// TIA Portal V16 export
// export: Created 2022-08-05T16:49:58.9120399Z, ExportSetting WithDefaults, DisplayName Totally Integrated Automation Portal, DisplayVersion V16, DisplayName TIA Portal Version Control Interface, DisplayVersion V16, DisplayName TIA Portal Openness, DisplayVersion V16, DisplayName SINAMICS Startdrive Advanced, DisplayVersion V16, DisplayName SINAMICS Startdrive G130, G150, S120, S150, SINAMICS MV, S210, DisplayVersion V16, DisplayName SINAMICS Startdrive G110M, G120, G120C, G120D, G120P, DisplayVersion V16, DisplayName STEP 7 Professional, DisplayVersion V16, DisplayName STEP 7 Safety, DisplayVersion V16, DisplayName WinCC Professional, DisplayVersion V16
VAR_GLOBAL   // PLC tag table "PuShButton_Interlocking"
   Stop AT %I0.0 : Bool;
   Forward_Start AT %I0.1 : Bool;
   Forward_Motor AT %Q0.0 : Bool;
   Back_Start AT %I0.2 : Bool;
   Back_Motor AT %Q0.1 : Bool;
END_VAR
